// TIA Portal V19 export
DATA_BLOCK "A0301_Spintore_Lat"   // DB121
// stored: InstanceOfName A0301_Spintore_Lat_FB, InstanceOfType FB
"A0301_Spintore_Lat_FB"
   // VAR_INPUT
   //    AreaInterface { ExternalAccessible := 'False'; ExternalVisible := 'False'; ExternalWritable := 'False'} : "AreaInterface";
   //    ZSI { ExternalAccessible := 'False'; ExternalVisible := 'False'; ExternalWritable := 'False'} : "udt_ZoneSafetyInterface";
   //    DSI { ExternalAccessible := 'False'; ExternalVisible := 'False'; ExternalWritable := 'False'} : "udt_DeviceSafetyInterface";
   //    DataIn : Struct
   //       OP_Rest_PB : Bool;
   //       OP_Work_PB : Bool;
   //       Orz_1_AnalSens : Int;
   //       Orz_2_AnalSens : Int;
   //    END_STRUCT;
   //    CIn { ExternalAccessible := 'False'; ExternalVisible := 'False'; ExternalWritable := 'False'} : Struct
   //       Manager_SpinLat_1 : "ValveMachine_Manager";
   //       Manager_SpinLat_2 : "ValveMachine_Manager";
   //       Manager_Sollevatori : "ValveMachine_Manager";
   //       SemiAut_Pb : Bool;
   //       P4 : Struct
   //          Fermi : "ValveMachine_COut";
   //       END_STRUCT;
   //       P5 : Struct
   //          SpintoreLong : Struct
   //             Ax_Sts : Struct
   //                PosAttesa_Reached : Bool;
   //                PosFineSpinta_Reached : Bool;
   //             END_STRUCT;
   //             Spintore : "ValveMachine_COut";
   //             Ax : "Positioning_EPOS_Machine_COut";
   //             Vrt : "ValveMachine_COut";
   //             Orz : "ValveMachine_COut";
   //          END_STRUCT;
   //       END_STRUCT;
   //       Trasporto : "SpeedMachine_COut";
   //    END_STRUCT;
   //    Config : Struct
   //       Vrt_1 : "ValveMachine_Config";
   //       Orz_1 : "ValveMachine_Config";
   //       Vrt_2 : "ValveMachine_Config";
   //       Orz_2 : "ValveMachine_Config";
   //       Sollevatori : Array[1..7] of "ValveMachine_Config";
   //       QuotaIngombro_SpinLat2 : Real;
   //       QuotaIngombro_SpinLat1 { ExternalWritable := 'False'} : Real;
   //       DelayMissingCondition : Time;
   //    END_STRUCT;
   // END_VAR
   // VAR_OUTPUT
   //    MachineInterface : "MachineInterface";
   //    COut : Struct
   //       Spin_Lat1 : Struct
   //          Standstill : Bool;
   //          Rest_CheckNext : Bool;
   //          Work_CheckNext : Bool;
   //          Rest : Bool;
   //          Work : Bool;
   //       END_STRUCT;
   //       Spin_Lat2 : Struct
   //          Standstill : Bool;
   //          Rest_CheckNext : Bool;
   //          Work_CheckNext : Bool;
   //          Rest : Bool;
   //          Work : Bool;
   //       END_STRUCT;
   //       Vrt_1 : "ValveMachine_COut";
   //       Orz_1 : "ValveMachine_COut";
   //       Vrt_2 : "ValveMachine_COut";
   //       Orz_2 : "ValveMachine_COut";
   //       Sollevatori : "ValveMachine_COut";
   //    END_STRUCT;
   // END_VAR
   // VAR_IN_OUT
   //    Spin_Lat_1 : Struct
   //       Par : "Analogic_SensorManagement_Par";
   //       Data : Struct
   //          Sens : "Analogic_SensorManagement_Data";
   //          HMI : "HMI_Preset";
   //       END_STRUCT;
   //       Par_Mach : "A0301_Mach_Sens_Par";
   //    END_STRUCT;
   //    Spin_Lat_2 : Struct
   //       Par : "Analogic_SensorManagement_Par";
   //       Data : Struct
   //          Sens : "Analogic_SensorManagement_Data";
   //          HMI : "HMI_Preset";
   //       END_STRUCT;
   //       Par_Mach : "A0301_Mach_Sens_Par";
   //    END_STRUCT;
   // END_VAR
   // VAR
   //    Alarm : Struct
   //       Vrt_1 : "ValveAlr";
   //       Orz_1 { S7_SetPoint := 'True'} : "ValveAlr";
   //       Orz_1_AnalSens_Issue : Bool;
   //       Vrt_2 : "ValveAlr";
   //       Orz_2 { S7_SetPoint := 'True'} : "ValveAlr";
   //       Orz_2_AnalSens_Issue : Bool;
   //       Sollevatori : Array[1..7] of "ValveAlr";
   //       Finestre : Struct
   //          SpinLat2_SpinLong_Stop : Bool;
   //          SpinLat1_SpinLong_Stop : Bool;
   //       END_STRUCT;
   //    END_STRUCT;
   //    Warning : Struct
   //       Vrt_1 : "ValveMachine_Wng";
   //       Orz_1 { S7_SetPoint := 'True'} : "ValveMachine_Wng";
   //       Orz_1_AnalSens { ExternalAccessible := 'False'; ExternalVisible := 'False'; ExternalWritable := 'False'} : "Analogic_SensorManagement_Warning";
   //       Vrt_2 : "ValveMachine_Wng";
   //       Orz_2 { S7_SetPoint := 'True'} : "ValveMachine_Wng";
   //       Orz_2_AnalSens { ExternalAccessible := 'False'; ExternalVisible := 'False'; ExternalWritable := 'False'} : "Analogic_SensorManagement_Warning";
   //       Sollevatori : Array[1..7] of "ValveMachine_Wng";
   //       Finestre : Struct
   //          SpinLat2_SpinLong_Stop : Bool;
   //          SpinLat1_SpinLong_Stop : Bool;
   //       END_STRUCT;
   //       OP_REST_MissingCnd : Bool;
   //       OP_WORK_MissingCnd : Bool;
   //    END_STRUCT;
   //    HMI : Struct
   //       Selection : Array[1..6] of Bool;
   //       Sollevatori_Sts { S7_SetPoint := 'True'} : "UDT_HMI-Sts_ValvePosA0301";
   //       "SpinLat1&2_Sts" { S7_SetPoint := 'True'} : "UDT_HMI-Sts_ValvePosA0301";
   //       "SpinLat1&2_Vrt_Sts" { S7_SetPoint := 'True'} : "UDT_HMI-Sts_ValvePosA0301";
   //       "SpinLat1&2_Orz_Sts" { S7_SetPoint := 'True'} : "UDT_HMI-Sts_ValvePosA0301";
   //       Orz_AnalSens_PB_Preset { ExternalAccessible := 'False'; ExternalVisible := 'False'; ExternalWritable := 'False'} : Bool;
   //       Orz_AnalSens_Preset_Value : LReal;
   //    END_STRUCT;
   //    Sts : Struct
   //       "SpinLat1&2_Alarm" : Bool;
   //       "SpinLat1&2_Vrt_AlarmPresence" : Bool;
   //       "SpinLat1&2_Orz_AlarmPresence" : Bool;
   //       Sollevatori_AlarmPresence : Bool;
   //       OP_CanMoveFreely : Bool;
   //       OP_Rest_Cnd : Bool;
   //       Op_Work_Cnd : Bool;
   //       Beam : Struct
   //          H_B : Real;
   //          Len_Meas : Real;
   //          P_U_PLen : Real;
   //          P_L_PLen : Real;
   //       END_STRUCT;
   //       "En/Dis_SpinLat_2" : Bool := TRUE;
   //    END_STRUCT;
   //    Ctrl : Struct
   //       OP_Rest_Man : Bool;
   //       OP_Work_Man : Bool;
   //       OP_Rest_Aut : Bool;
   //       OP_Work_Aut : Bool;
   //       OP_Rest : Bool;
   //       OP_Work : Bool;
   //    END_STRUCT;
   //    Vrt_1 : "ValveMachine_FB";
   //    Orz_1 { S7_SetPoint := 'True'} : "ValveMachine_FB";
   //    Orz_1_AnalSens { S7_SetPoint := 'True'} : "Analogic_SensorManagement";
   //    Vrt_2 : "ValveMachine_FB";
   //    Orz_2 { S7_SetPoint := 'True'} : "ValveMachine_FB";
   //    Orz_2_AnalSens { S7_SetPoint := 'True'} : "Analogic_SensorManagement";
   //    Sollevatori : Array[1..6] of "ValveMachine_FB";
   //    AUX : Struct
   //       OP_Rest_PB : Bool;
   //       OP_Work_PB : Bool;
   //    END_STRUCT;
   //    TON_OP_REST_MissingCnd { S7_SetPoint := 'True'} : TON_TIME;
   //    TON_OP_WORK_MissingCnd { S7_SetPoint := 'True'} : TON_TIME;
   //    Finestre : Struct
   //       Quota_SpinLat2_Rest : Real := 2705.0;
   //       Quota_SpinLat1_Rest : Real := 4000.0;
   //       RestCnd_Vrt_1 : Bool;
   //       RestCnd_Vrt_2 : Bool;
   //    END_STRUCT;
   // END_VAR
BEGIN
   HMI.Selection[1..6] := TRUE;
END_DATA_BLOCK
